// TIA Portal V20 export
FUNCTION "LER_stepStatusFC" : Void   // FC75, LAD
// stored: Access Published, SetENOAutomatically false
   VAR_INPUT
      emName : String;
      enabled : Bool;
      initialized : Bool;
      active : Bool;
      complete : Bool;
      currentStep : DInt;
      stepCommand : "LER_typeStep";
   END_VAR
   VAR_OUTPUT
      hmiStepStatus : "LER_typeAutoStep";
   END_VAR
   VAR_TEMP   // added for the SCL form of the ladder/FBD networks
      _w1 : Bool;
      _w2 : Bool;
   END_VAR
BEGIN

REGION Network 2 (SCL): Name
   #hmiStepStatus.emNameString := #emName;
END_REGION

REGION Network 3: Status
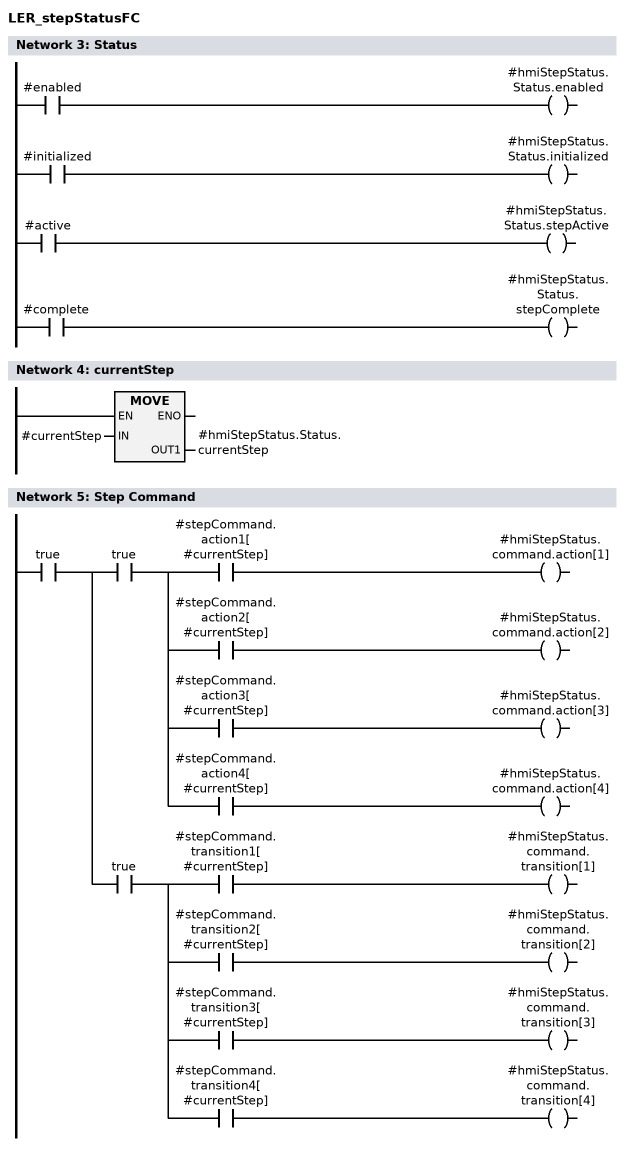
   RUNG wire#powerrail
      Contact( #enabled )
      Coil( #hmiStepStatus.Status.enabled )
   END_RUNG
   RUNG wire#powerrail
      Contact( #initialized )
      Coil( #hmiStepStatus.Status.initialized )
   END_RUNG
   RUNG wire#powerrail
      Contact( #active )
      Coil( #hmiStepStatus.Status.stepActive )
   END_RUNG
   RUNG wire#powerrail
      Contact( #complete )
      Coil( #hmiStepStatus.Status.stepComplete )
   END_RUNG
   // the same network as SCL:
   #hmiStepStatus.Status.enabled := #enabled;
   #hmiStepStatus.Status.initialized := #initialized;
   #hmiStepStatus.Status.stepActive := #active;
   #hmiStepStatus.Status.stepComplete := #complete;
END_REGION

REGION Network 4: currentStep
   RUNG wire#powerrail
      Move(in := #currentStep, out1 => #hmiStepStatus.Status.currentStep)
   END_RUNG
   // the same network as SCL:
   #hmiStepStatus.Status.currentStep := #currentStep;
END_REGION

REGION Network 5: Step Command
   RUNG wire#powerrail
      Contact( true )
      wire#w1
      Contact( true )
      wire#w2
      Contact( #stepCommand.action1[#currentStep] )
      Coil( #hmiStepStatus.command.action[1] )
   END_RUNG
   RUNG wire#w2
      Contact( #stepCommand.action2[#currentStep] )
      Coil( #hmiStepStatus.command.action[2] )
   END_RUNG
   RUNG wire#w2
      Contact( #stepCommand.action3[#currentStep] )
      Coil( #hmiStepStatus.command.action[3] )
   END_RUNG
   RUNG wire#w2
      Contact( #stepCommand.action4[#currentStep] )
      Coil( #hmiStepStatus.command.action[4] )
   END_RUNG
   RUNG wire#w1
      Contact( true )
      wire#w3
      Contact( #stepCommand.transition1[#currentStep] )
      Coil( #hmiStepStatus.command.transition[1] )
   END_RUNG
   RUNG wire#w3
      Contact( #stepCommand.transition2[#currentStep] )
      Coil( #hmiStepStatus.command.transition[2] )
   END_RUNG
   RUNG wire#w3
      Contact( #stepCommand.transition3[#currentStep] )
      Coil( #hmiStepStatus.command.transition[3] )
   END_RUNG
   RUNG wire#w3
      Contact( #stepCommand.transition4[#currentStep] )
      Coil( #hmiStepStatus.command.transition[4] )
   END_RUNG
   // the same network as SCL:
   #_w1 := true AND true;
   #hmiStepStatus.command.action[1] := #_w1 AND #stepCommand.action1[#currentStep];
   #hmiStepStatus.command.action[2] := #_w1 AND #stepCommand.action2[#currentStep];
   #hmiStepStatus.command.action[3] := #_w1 AND #stepCommand.action3[#currentStep];
   #hmiStepStatus.command.action[4] := #_w1 AND #stepCommand.action4[#currentStep];
   #_w2 := true AND true;
   #hmiStepStatus.command.transition[1] := #_w2 AND #stepCommand.transition1[#currentStep];
   #hmiStepStatus.command.transition[2] := #_w2 AND #stepCommand.transition2[#currentStep];
   #hmiStepStatus.command.transition[3] := #_w2 AND #stepCommand.transition3[#currentStep];
   #hmiStepStatus.command.transition[4] := #_w2 AND #stepCommand.transition4[#currentStep];
END_REGION
END_FUNCTION
